// Mitsubishi GX Works2 project: basic_operations   PLC: Q03UDV

PROGRAM MAIN
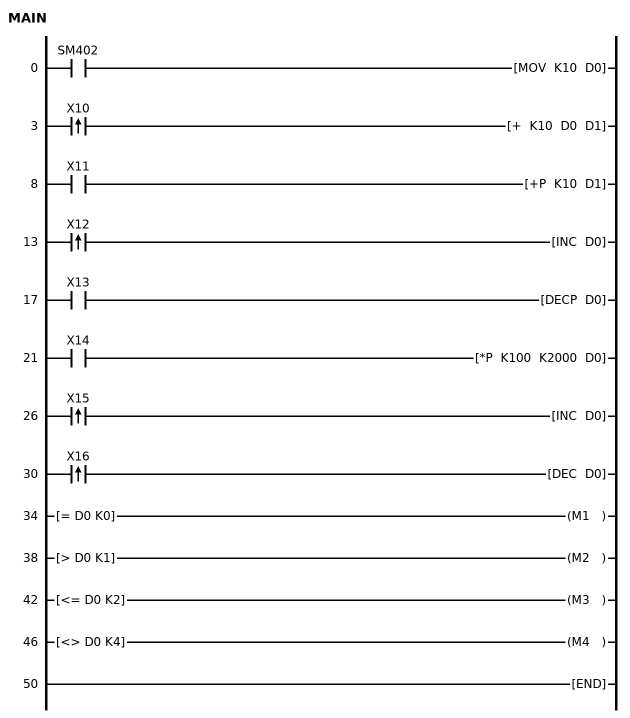
0     LD      SM402
      MOV     K10 D0
3     LDP     X10
      +       K10 D0 D1
8     LD      X11
      +P      K10 D1
13    LDP     X12
      INC     D0
17    LD      X13
      DECP    D0
21    LD      X14
      *P      K100 K2000 D0
26    LDP     X15
      INC     D0
30    LDP     X16
      DEC     D0
34    LD=     D0 K0
      OUT     M1
38    LD>     D0 K1
      OUT     M2
42    LD<=    D0 K2
      OUT     M3
46    LD<>    D0 K4
      OUT     M4
50    END
END_PROGRAM
